# EPICS StreamDevice protocol: db/hallprobe.proto
Terminator = LF;
ReplyTimeout = 2000;
ReadTimeout = 1000;

readField {
    ExtraInput = Ignore;
    in "%f";
}
